# EPICS substitutions: mc11/db/pmacStatus.substitutions
file "db/pmacStatus.db"
{
pattern
{SYS,             PMAC,    VERSION  PLC  PORT,  NAXES }
{"XF:23ID2-CT",   "MC:11",  "1"      5    "P0",  8     }
}
